KUKA KRL data list: OscilationTest.dat

&ACCESS RVP
&REL 1
DEFDAT OscilationTest PUBLIC

ENDDAT
